(* IEC 61131-3 sources: LLM-CodeGen-RAG/OpenPLC, 2 files *)

(* ---- sh1.st ---- *)
FUNCTION_BLOCK fb_SampleAndAverage
VAR_INPUT
    Signal_In: REAL;
    PT: TIME := T#1s;
    N: INT := 8;
END_VAR

VAR_OUTPUT
    AVG: REAL;
END_VAR

VAR
    fb_SH_1: SH_1;
    fb_FT_AVG: FT_AVG;
END_VAR

fb_SH_1(IN := Signal_In, PT := PT);
fb_FT_AVG(IN := fb_SH_1.OUT, N := N);
AVG := fb_FT_AVG.OutputREAL;
END_FUNCTION_BLOCK

(* ---- sine.st ---- *)
FUNCTION_BLOCK SINE_TO_STAIR
VAR_INPUT
END_VAR
VAR_OUTPUT
  outputSignal: REAL;
END_VAR
VAR
  genSin: GEN_SIN;
  stair: STAIR;
END_VAR
genSin(PT := T#10S, AM := 10, OS := 5, DL := 0);
stair(X := genSin.OUT, D := 2.3);
outputSignal := stair.OUTPUT;
END_FUNCTION_BLOCK
